PROGRAM PRG_SafetyLightCurtain
VAR
END_VAR

GVL.bSafeRedLedOutput := GVL.bSafeRedLedInput;
GVL.bSafeRestartSignal:=GVL.bSafeRestartSignalInput;

END_PROGRAM

(* stored: Version 1.1.0.1, ProductVersion 3.1.4024.12
   POU PRG_SafetyLightCurtain: Id {9fc58935-82cf-401e-98fd-fe4f9b763d73}, SpecialFunc None *)
